FUNCTION_BLOCK Conveyor EXTENDS A_Actuator

VAR_OUTPUT
	bForward  : BOOL;
	bBackward  : BOOL;
END_VAR

VAR	
	fbForward : BoolOut;
	fbBackward : BoolOut;
END_VAR

super^();
bForward := fbForward.getValue;
bBackward := fbBackward.getValue;

METHOD backward : BOOL
VAR_INPUT
END_VAR
fbForward.setValue := FALSE;
fbBackward.setValue := TRUE;
END_METHOD

METHOD  executeCmd : BOOL
VAR_INPUT
	
END_VAR
SUPER^.executeCmd();

CASE eCmd OF
	eFORWARD:
		forward();
	eBACKWARD:
		backward();
END_CASE
END_METHOD

METHOD forward : BOOL
VAR_INPUT
END_VAR
fbForward.setValue := TRUE;
fbBackward.setValue := FALSE;
END_METHOD

PROPERTY getBackward : I_StepCondition
GET
getBackward := fbBackward;
END_GET
END_PROPERTY

PROPERTY getForward : I_StepCondition
GET
getForward := fbForward;
END_GET
END_PROPERTY

END_FUNCTION_BLOCK

(* stored: Version 1.1.0.1, ProductVersion 3.1.4024.2
   POU Conveyor: Id {b15311d8-a9f4-4077-9cec-ef51ff0c9999}, SpecialFunc None
   Method backward: Id {60abf0c4-e96b-4752-92c0-f03aac1192c2}
   Method executeCmd: Id {abede58c-7ad4-4264-be60-72700c8f52b7}
   Method forward: Id {814a72d6-f33d-43b0-a610-4157c76afd05}
   Property getBackward: Id {7ca234ea-7c61-4075-89ec-893e796ebe8c}
   Get Get: Id {e25e64f7-4659-4a1b-9897-d675065c8e35}
   Property getForward: Id {6370b0c0-d40e-456d-89ce-6f31c418ed60}
   Get Get: Id {489b8359-b98c-42ae-afe2-3461bd22238e} *)
